FUNCTION_BLOCK T_PulseTimer
VAR
    TP1 : TP;
END_VAR

METHOD FB_init : BOOL
VAR_INPUT
    bInitRetains : BOOL;  // if TRUE, the retain variables are initialized (warm start / cold start)
    bInCopyCode  : BOOL;  // if TRUE, the instance afterwards gets moved into the copy code (online change)
    PresetTime   : LREAL; // seconds
END_VAR
TP1.PT := LREAL_TO_TIME(PresetTime * 1000);
END_METHOD

PROPERTY OutputState : BOOL
GET
OutputState := TP1.Q;
END_GET
END_PROPERTY

PROPERTY PresetTime : LREAL
GET
PresetTime := TIME_TO_LREAL(TP1.PT) / 1000.0; // in seconds
END_GET
SET
TP1.PT := LREAL_TO_TIME(PresetTime * 1000);
END_SET
END_PROPERTY

METHOD Pulse : BOOL
VAR_INPUT
    In : BOOL;
END_VAR
TP1(IN := In);
Pulse := TP1.Q;
END_METHOD

METHOD Reset
TP1(IN := FALSE);
END_METHOD

METHOD Run : BOOL
TP1(IN := TRUE);
Run := TP1.Q;
END_METHOD

END_FUNCTION_BLOCK

(* stored: Version 1.1.0.1, ProductVersion 3.1.4024.12
   POU T_PulseTimer: Id {c0de455d-de15-4ff4-bb4a-84dda6f6beaa}, SpecialFunc None
   Method FB_init: Id {4d6ab5ac-dd98-486d-a60c-5ce9af0f2917}
   Property OutputState: Id {c7de3cbe-20f0-48e2-86ea-50cc524cc1a0}
   Get Get: Id {e72204b1-24bd-4fa6-bba6-739301d18e97}
   Property PresetTime: Id {e8c4b05a-61b1-4127-b4b5-d0535e759a21}
   Get Get: Id {48846de1-b0fe-4ab7-9c13-2694bd1509eb}
   Set Set: Id {0593ca43-9469-42c1-8110-c4385f6b0287}
   Method Pulse: Id {5fecae55-d662-44eb-a1d7-deb30dba60ed}
   Method Reset: Id {6a9bf7c8-fac5-454a-8eb0-e6cf5daae26c}
   Method Run: Id {7853bc9f-a157-40e6-a9ee-cfe54ad6f258} *)
